PROGRAM MAIN
VAR 
	
END_VAR

END_PROGRAM

(* stored: Version 1.1.0.1, ProductVersion 3.1.4024.12
   POU MAIN: Id {9e56dcee-d0d6-48bd-9509-377001e6a204}, SpecialFunc None *)
